% RSLogix 500 project P3_ABIOLA_A_V15 BRANCHED_BAK084.RSS, saved by version 8.30.00.16 %
PROJECT "UNTITLED"    % processor: Bul.1763 MicroLogix 1100 Series B %

PROGRAM FILES
  LAD 2   2 rungs
  LAD 3 "PSEUDO IO"  19 rungs  % Contains all the assigned memery address used  %

DATA FILES
  O0 OUTPUT  4 elements
  I1 INPUT  6 elements
  S2 STATUS  66 elements
  B3 BINARY  1 elements
  T4 TIMER  1 elements
  C5 COUNTER  1 elements
  R6 CONTROL  1 elements
  N7 INTEGER  11 elements
  F8 FLOAT  1 elements
  ST9 STRFRBCSCN  20 elements  % Writes string from bar code scanner to PLC %
  ST10 STRING  10 elements

LADDER 2
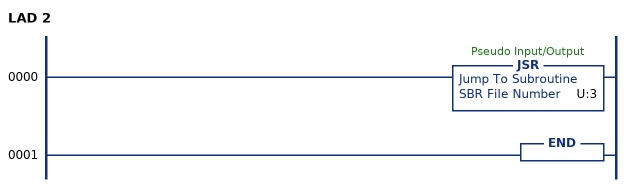
% Rung: 0 %
SOR JSR U:3 EOR
%   U:3  "Pseudo Input/Output" %
% Rung: 1 %
SOR END EOR

LADDER 3 "PSEUDO IO"    % Contains all the assigned memery address used  %
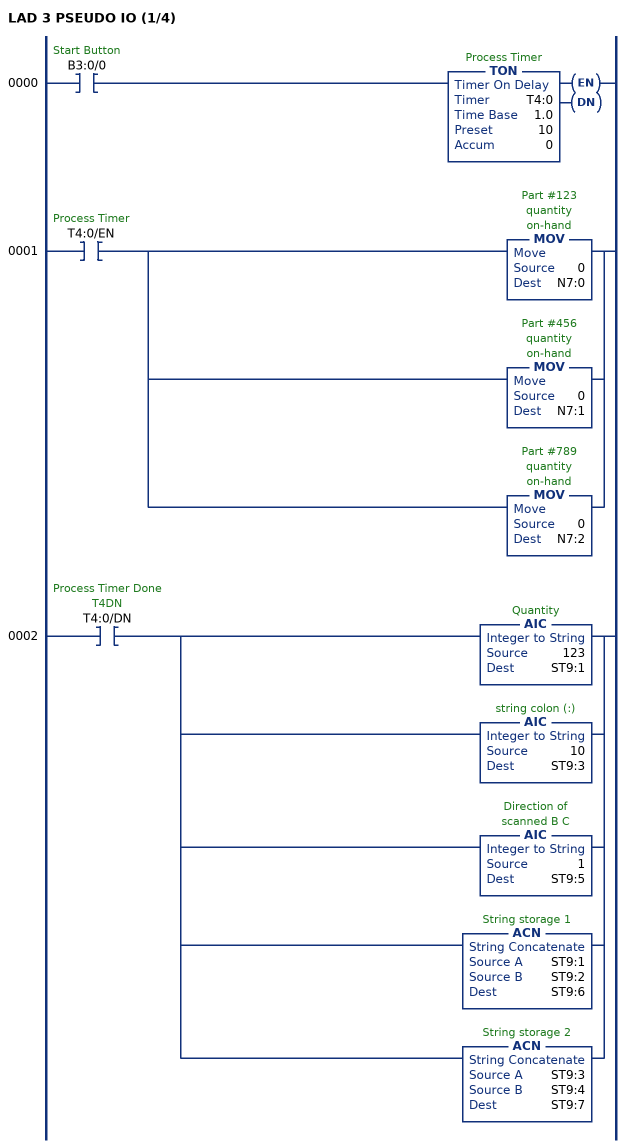
% Rung: 0 %
SOR XIC B3:0/0 TON T4:0 1.0 10 0 EOR
%   B3:0/0  "Start Button" %
%   T4:0  "Process Timer" %
% Rung: 1 %
SOR XIC T4:0/EN BST MOV 0 N7:0 NXB BST MOV 0 N7:1 NXB MOV 0 N7:2 BND BND EOR
%   T4:0  "Process Timer" %
%   N7:0  "Part #123 quantity on-hand" %
%   N7:1  "Part #456 quantity on-hand" %
%   N7:2  "Part #789 quantity on-hand" %
% Rung: 2 %
SOR XIC T4:0/DN BST AIC 123 ST9:1 NXB BST AIC 10 ST9:3 NXB BST AIC 1 ST9:5 NXB BST ACN ST9:1 ST9:2 ST9:6 NXB ACN ST9:3 ST9:4 ST9:7 BND BND BND BND EOR
%   T4:0/DN  T4DN  "Process Timer Done" %
%   ST9:1  "Quantity" %
%   ST9:3  "string colon (:)" %
%   ST9:5  "Direction of scanned B C" %
%   ST9:2  "String Quantity from Bar-code scanner" %
%   ST9:6  "String storage 1" %
%   ST9:4  "Concatination of colon (:) with direction from BCS" %
%   ST9:7  "String storage 2" %

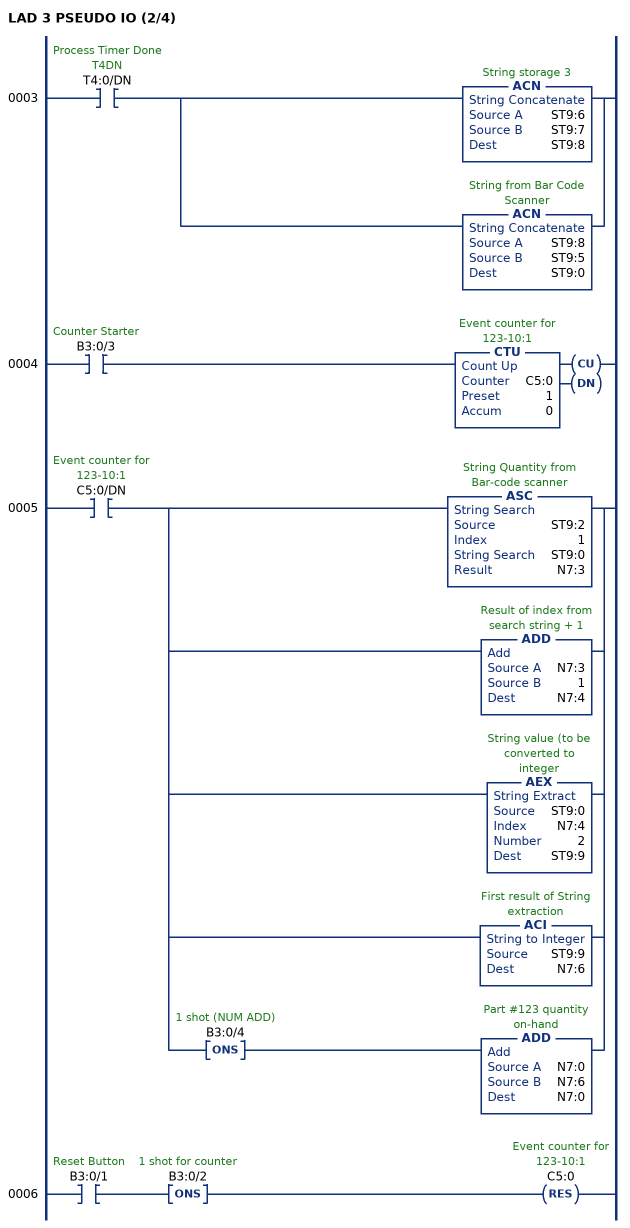
% Rung: 3 %
SOR XIC T4:0/DN BST ACN ST9:6 ST9:7 ST9:8 NXB ACN ST9:8 ST9:5 ST9:0 BND EOR
%   T4:0/DN  T4DN  "Process Timer Done" %
%   ST9:6  "String storage 1" %
%   ST9:7  "String storage 2" %
%   ST9:8  "String storage 3" %
%   ST9:5  "Direction of scanned B C" %
%   ST9:0  "String from Bar Code Scanner" %
% Rung: 4 %
SOR XIC B3:0/3 CTU C5:0 1 0 EOR
%   B3:0/3  "Counter Starter" %
%   C5:0  "Event counter for 123-10:1" %
% Rung: 5 %
SOR XIC C5:0/DN BST BST ASC ST9:2 1 ST9:0 N7:3 NXB ADD N7:3 1 N7:4 BND NXB BST AEX ST9:0 N7:4 2 ST9:9 NXB BST ACI ST9:9 N7:6 NXB ONS B3:0/4 ADD N7:0 N7:6 N7:0 BND BND BND EOR
%   C5:0  "Event counter for 123-10:1" %
%   ST9:2  "String Quantity from Bar-code scanner" %
%   ST9:0  "String from Bar Code Scanner" %
%   N7:3  "Constant value of 10" %
%   N7:4  "Result of index from search string + 1" %
%   ST9:9  "String value (to be converted to integer" %
%   N7:6  "First result of String extraction" %
%   B3:0/4  "1 shot (NUM ADD)" %
%   N7:0  "Part #123 quantity on-hand" %
% Rung: 6 %
SOR XIC B3:0/1 ONS B3:0/2 RES C5:0 EOR
%   B3:0/1  "Reset Button" %
%   B3:0/2  "1 shot for counter" %
%   C5:0  "Event counter for 123-10:1" %

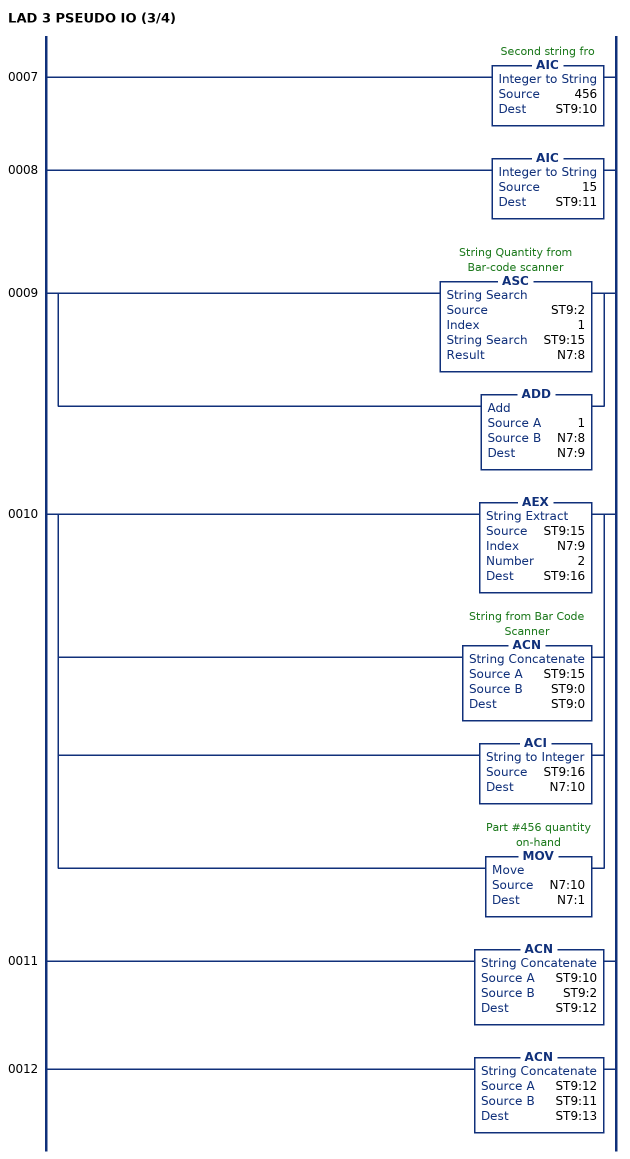
% Rung: 7 %
SOR AIC 456 ST9:10 EOR
%   ST9:10  "Second string fro" %
% Rung: 8 %
SOR AIC 15 ST9:11 EOR
% Rung: 9 %
SOR BST ASC ST9:2 1 ST9:15 N7:8 NXB ADD 1 N7:8 N7:9 BND EOR
%   ST9:2  "String Quantity from Bar-code scanner" %
% Rung: 10 %
SOR BST BST AEX ST9:15 N7:9 2 ST9:16 NXB ACN ST9:15 ST9:0 ST9:0 BND NXB BST ACI ST9:16 N7:10 NXB MOV N7:10 N7:1 BND BND EOR
%   ST9:0  "String from Bar Code Scanner" %
%   N7:1  "Part #456 quantity on-hand" %
% Rung: 11 %
SOR ACN ST9:10 ST9:2 ST9:12 EOR
%   ST9:10  "Second string fro" %
%   ST9:2  "String Quantity from Bar-code scanner" %
% Rung: 12 %
SOR ACN ST9:12 ST9:11 ST9:13 EOR

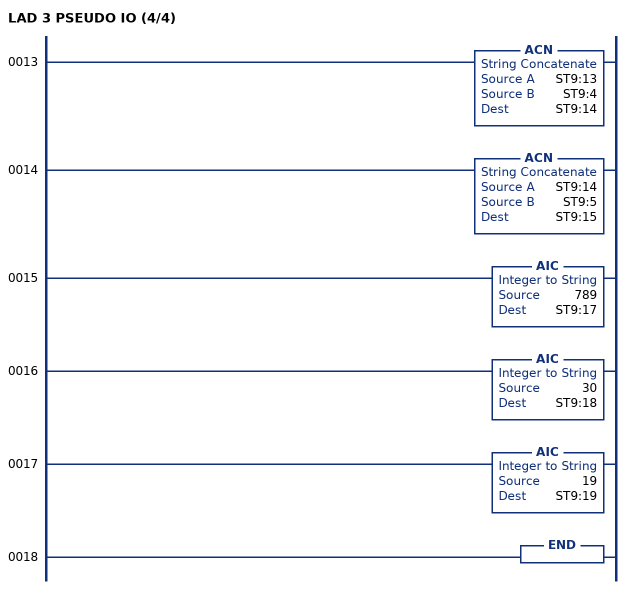
% Rung: 13 %
SOR ACN ST9:13 ST9:4 ST9:14 EOR
%   ST9:4  "Concatination of colon (:) with direction from BCS" %
% Rung: 14 %
SOR ACN ST9:14 ST9:5 ST9:15 EOR
%   ST9:5  "Direction of scanned B C" %
% Rung: 15 %
SOR AIC 789 ST9:17 EOR
% Rung: 16 %
SOR AIC 30 ST9:18 EOR
% Rung: 17 %
SOR AIC 19 ST9:19 EOR
% Rung: 18 %
SOR END EOR

OTHER DOCUMENTED ADDRESSES
  C5:0.ACC  "Number of count storage"
  C5:0/CU  "Process counter"
  N7:5  "String colon (:) converted to integer"
  ST9:2.0  "Result of Constant Multiplication with -1"
  ST10:1.0  "String len"

DATA TABLE (non-zero values as saved)
DATA T4
% .PRE .ACC %
% T4:0 % 10 0
DATA C5
% .PRE .ACC %
% C5:0 % 1 0
DATA ST9
% ST9:0 % "\00\00\00\00\00\00\00\00"
% ST9:2 % "-"
% ST9:4 % ":"
